TYPE T_Ctrl_SIf_ICL_Cfg :
STRUCT
	Module: T_Ctrl_SIf_MOD_Cfg;
END_STRUCT
END_TYPE

(* stored: Version 1.1.0.1, ProductVersion 3.1.0.19
   DUT T_Ctrl_SIf_ICL_Cfg: Id {e06885a1-5b91-4de5-ac45-d80962cde19e} *)
